# EPICS substitutions: ecmcApp/Db/SlitX-xp-extra.substitutions
file "ecmc-extra.template"
{
pattern
{P,      M,    R,   PORT, ADDR, PREC, HOMEPROC}
{IOC2:,  xp, xp-,   MCU1,    1, 3,    3}
}
